Universal Robots PolyScope program: followerUR10e.urp

Program followerUR10e (installation=followerUR10e directory=/programs/usbdisk/leaderFollower createdIn=5.12.4 lastSavedIn=5.23.0 robotSerialNumber=20195000937)
Calibrated DH parameters: a=[0.000264, -0.612377, -0.484433, 0.000064, -0.000025, 0]; d=[0.180726, -15.534777, 180.69926, -164.989927, 0.119929, 0.115635]; alpha=[1.570213, 0.000851, -0.001835, 1.570844, -1.57144, 0]; deltaTheta=[0, -0.02159, -0.537544, 0.559142, 0.000001, 0]
InitVariablesNode
BeforeStart
  Popup Message (haltProgram=false message=Remember to set the Leader robots ip in the Installation->Fieldbus->Modbus settings inputType=Text)
  Script file /programs/usbdisk/booth_programs/ERF2023/general.script
    | PI = acos(-1)
    | PI2 = PI*2
    | mPI = PI*1000
    | mPI2 = PI2*1000
    | 
    | def unsignedToSigned(i):
    |   if i > 32767:
    |     return i - 65536
    |   end
    |   return i
    | end
    | 
    | firstGetAngle = True
    | def getAngle(rev,angle, last):
    |   r=unsignedToSigned(rev)
    |   new = r*PI2 + angle/1000
    | 
    |   if norm(new - last) > 1 and not firstGetAngle:
    |     return last
    |   end
    | 
    |   return new
    | end
    | 
    | def mirror(j):
    |   return j * [-1,-1,-1,-1,-1,-1]+ [0,-PI,0,-PI,0,0]
    | end
    | 
    | def maxDiff(a,b, limit):
    |   global abNorm = norm(a-b)
    |   return abNorm < limit
    | end
  last_go := get_target_joint_positions()
  ur1 := get_target_joint_positions()
  doMirror :=  (valueSource=Operator message=Mirror mode? valueType=Boolean)
Robot Program (runOnlyOnce=false)
  ur1 := [getAngle(baseR,base,ur1[0]), getAngle(shoulderR,shoulder, ur1[1]), getAngle(elbowR,elbow, ur1[2]), getAngle(wrist1R,wrist1,ur1[3]), getAngle(wrist2R,wrist2,ur1[4]), getAngle(wrist3R,wrist3,ur1[5])]
  Script: firstGetAngle =  False
  If doMirror
    go := mirror(ur1)
  Else 
    go := ur1
  Script: sync()
  last_go := go
Thread Thread_1 (runOnlyOnce=false)
  initLimit := 0.1
  Loop While (checkContinuously=false) expression=not maxDiff(last_go, get_target_joint_positions(), initLimit)
    MoveJ speed 10 deg/s, acceleration 80 deg/s^2 (useActiveTCP=true positionType=JointAngles optimoveEnabled=false optiMoveSpeed=0.3 optiMoveAcceleration=0.09) feature=Base
      Waypoint Variable (Variable): variable=go
  initLimit := 0.5
  Loop While (checkContinuously=true) expression=maxDiff(last_go, get_target_joint_positions(), initLimit)
    Script: servoj(go, 2, t=get_steptime(), lookahead_time=0.05, gain=500)
